{attribute 'qualified_only'}
{attribute 'strict'}
TYPE stIOSensorTypes :
(
	AI_4To20ma := 0,
	AI_PT100	:= 1,
	AI_0To10V	:=2,
	AI_0To5V	:=3
	
);
END_TYPE

(* stored: Version 1.1.0.1, ProductVersion 3.1.4024.11
   DUT stIOSensorTypes: Id {851dca04-9a8c-497e-9748-e34195cfdc8d} *)
